(* PLC project LearnCODESYS_1.project, CODESYS CODESYS V3.5 SP21 Patch 3 *)
(* stored: creationDateTime 2026-05-28T15:03:11.8278016, modificationDateTime 2026-01-26T14:31:29.3036688 *)

FUNCTION_BLOCK myFBD
  VAR_OUTPUT
    outVar : DINT;
    x : BOOL;
  END_VAR
  VAR_INPUT
    newVar1 : DINT;
  END_VAR
  VAR CONSTANT
    tmp : DINT := 12;
  END_VAR
  VAR_INPUT
    newVar2 : DINT;
  END_VAR
  VAR
    t1 : BOOL;
    mnmn : ARRAY[1..5] OF BOOL;
  END_VAR

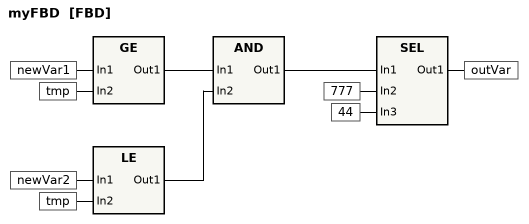
(* FBD diagram, written out as Structured Text *)
outVar := SEL(newVar1 >= tmp AND newVar2 <= tmp, 777, 44);
END_FUNCTION_BLOCK
